(* LS Electric XG5000 project: 241008_실습2깜박이펑션블록제작 *)
(* PLC LSPLC *)
(* module base 0 slot 0: 입력 모듈:XGI-D21A (DC 24V 입력, 8점 (전류소스/싱크입력)) *)
(* module base 0 slot 1: 출력 모듈:XGQ-RY1A (릴레이 출력, 8점 (2A용, 단독 COM.)) *)

FUNCTION_BLOCK ON_OFF
VAR_INPUT
    FL : BOOL;
    NFL : BOOL;
    OFF : BOOL;
END_VAR
VAR_OUTPUT
    LAMP1 : BOOL;
    LAMP2 : BOOL;
END_VAR
VAR
    T1 : TP;
    time5s : TIME := T#5s; (* 5초 동안 깜박 *)
END_VAR

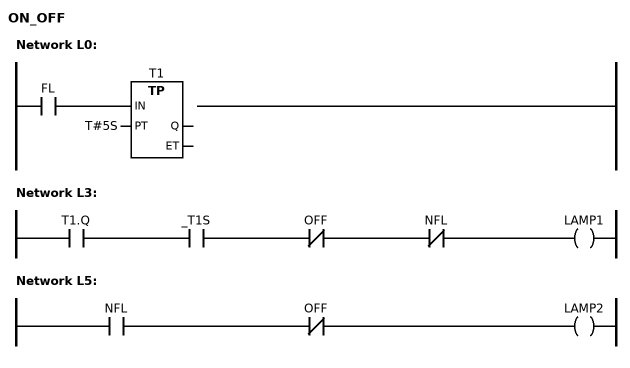
(* Rung L0 *)
T1(IN := FL, PT := T#5S);
(* Rung L3 *)
LAMP1 := T1.Q AND _T1S AND NOT OFF AND NOT NFL;
(* Rung L5 *)
LAMP2 := NFL AND NOT OFF;
END_FUNCTION_BLOCK

PROGRAM NewProgram (* task: 스캔 프로그램 *)
VAR
    OFF AT %IX0.0.3 : BOOL;
    ONON : ON_OFF;
    동작 : BOOL;
    램프 AT %QX0.1.0 : BOOL;
    램프2 AT %QX0.1.1 : BOOL;
    시작 AT %IX0.0.0 : BOOL;
    켜기 AT %IX0.0.1 : BOOL;
    켜기2 AT %IX0.0.2 : BOOL;
END_VAR

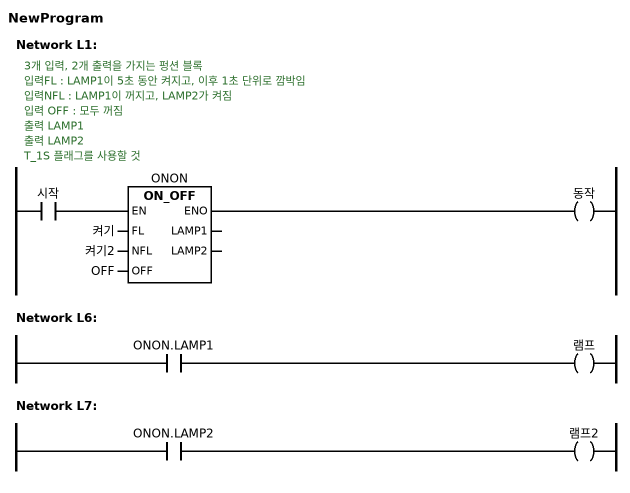
(* 3개 입력, 2개 출력을 가지는 펑션 블록 / 입력FL : LAMP1이 5초 동안 켜지고, 이후 1초 단위로 깜박임 / 입력NFL : LAMP1이 꺼지고, LAMP2가 켜짐 / 입력 OFF : 모두 꺼짐 / 출력 LAMP1 / 출력 LAMP2 / T_1S 플래그를 사용할 것 *)
(* Rung L1 *)
IF 시작 THEN ONON(FL := 켜기, NFL := 켜기2, OFF := OFF); END_IF;
동작 := 시작;
(* Rung L6 *)
램프 := ONON.LAMP1;
(* Rung L7 *)
램프2 := ONON.LAMP2;
END_PROGRAM